{attribute addProperty BoxType "EPP5101-0002-0016"}
{attribute addProperty Id "StatusAT %I*Status_B794ABE51621Counter_valueAT %I*UINT16217Latch_valueAT %I*UINT16218"}
{attribute addProperty CRC "417362543"}
{attribute addProperty SizeInBites "48"}
{attribute addProperty SizeInBytes "6"}
TYPE ENC_Status_compact_18E0726F :
STRUCT
	{attribute addProperty Name "Status"}
	Status AT %I* : Status_B794ABE5;
	{attribute addProperty Name "Counter_value"}
	Counter_value AT %I* : UINT;
	{attribute addProperty Name "Latch_value"}
	Latch_value AT %I* : UINT;
END_STRUCT
END_TYPE

(* stored: Version 1.2.0.0, ProductVersion 3.1.4024.9
   DUT ENC_Status_compact_18E0726F: Id {801ba539-f96a-4717-bde4-7a4bf4beb4d1} *)
